// TIA Portal V17 export
// export: Created 2023-12-22T15:04:39.9681609Z, ExportSetting WithDefaults, DisplayName Totally Integrated Automation Portal, DisplayVersion V17, DisplayName TIA Portal Openness, DisplayVersion V17, DisplayName TIA Portal Version Control Interface, DisplayVersion V17, DisplayName STEP 7 Professional, DisplayVersion V17, DisplayName STEP 7 Safety, DisplayVersion V17, DisplayName WinCC Advanced, DisplayVersion V17
FUNCTION_BLOCK "AI_ex"   // FB103, LAD
{ S7_Optimized_Access := 'FALSE' }
VERSION : 0.1
// stored: AutoNumber false, IsIECCheckEnabled false, SetENOAutomatically false, UDAEnableTagReadback false
   VAR_OUTPUT
      S_Alarm : Bool;   // Внешний индикатор наличия аварии
   END_VAR
   VAR_IN_OUT
      Signal : Int;   // Входной сигнал контроллера
      Result : Real;   // Результат измерений
   END_VAR
   VAR DB_SPECIFIC
      CMD : "CMD";   // Основные команды / Блок команд
      Mode : Int;   // Режим работы
      Status : Int;   // Статус устройства
      Use : Struct   // Функционал
         RTD { S7_SetPoint := 'True'} : Bool;   // Режим RTD
         Filter { S7_SetPoint := 'True'} : Bool;   // Филтрация сигнала
         Inverse { S7_SetPoint := 'True'} : Bool;   // Инверсия сигнала
         Indirect { S7_SetPoint := 'True'} : Bool := true;   // Косвенная адресация
         Status { S7_SetPoint := 'True'} : Bool;   // Использовать подсветку
         Light { S7_SetPoint := 'True'} : Bool;   // Динамическая подсветка
         Lim_Low { S7_SetPoint := 'True'} : Bool;   // Отсечь низкие аварии
         Lim_High { S7_SetPoint := 'True'} : Bool;   // Отсечь высокие аварии
         Communication { S7_SetPoint := 'True'} : Bool;   // Передача в Value по сети
      END_STRUCT;
      VmA : Real;   // Реальный сигнал на входе ПЛК
      RTD_c { S7_SetPoint := 'True'} : Real := 10.0;   // Коэффициент RTD
      Calibration { S7_SetPoint := 'True'} : Real;   // Поправка
   END_VAR
   VAR
      Converter { S7_SetPoint := 'True'} : "Converter_LAD";   // Масштабирование сигнала
   END_VAR
   VAR DB_SPECIFIC
      SP : Struct   // Уставки аварий
         NC { S7_SetPoint := 'True'} : Real := -500.0;   // Сигнал при обрыве линии
         SC { S7_SetPoint := 'True'} : Real := 32000.0;   // Сигнал при КЗ/перегрузке
         HH { S7_SetPoint := 'True'} : Real := 90.0;   // Аварийно высокий сигнал
         H { S7_SetPoint := 'True'} : Real := 85.0;   // Высокий сигнал
         L { S7_SetPoint := 'True'} : Real := 15.0;   // Низкий сигнал
         LL { S7_SetPoint := 'True'} : Real := 10.0;   // Аварийно низкий сигнал
      END_STRUCT;
   END_VAR
   VAR
      Tx { S7_SetPoint := 'True'} : Array[0..5] of "Time_R";   // Блок таймеров
   END_VAR
   VAR DB_SPECIFIC
      Alarm : Struct   // Список аварий
         ST : Bool;   // Общая неисправность
         HH : Bool;   // сработала авария по аварийно высокму уровню
         H : Bool;   // сработало предупреждение по высокому уровню
         L : Bool;   // сработало предупреждение по низкому уровню
         LL : Bool;   // сработало предупрждение по аварийно низкому уровню
         NC : Bool;   // обрыв линии
         SC : Bool;   // короткое замыкание
      END_STRUCT;
      Alarms : Word;   // Слово аварий
      Events : Word;   // События датчика
      pos : Array[0..15] of Bool;   // Контроль фронтов событий
      Input_Type { S7_SetPoint := 'True'} : Int;   // Тип датчика, 0 - 4..20, 1 - 0..20, 2 - 0..10, 3 - 0..5, 4 - RTD
      CodeID { S7_SetPoint := 'True'} : Int;   // Код датчика для привязки в скаде
      "Type" { S7_SetPoint := 'True'} : Int;   // Тип датчика (единицы измерения)
      ADDR { S7_SetPoint := 'True'} : Int;   // Адрес входа на контроллере
      Filter_SP { S7_SetPoint := 'True'} : Int := 100;   // Ёмкость фильтра
      "Name" { S7_SetPoint := 'True'} : String[5];
   END_VAR
   VAR
      Filter_DB : "Filter";   // Фильтрация скачков сигнала
   END_VAR
   VAR DB_SPECIFIC
      Time_DTL { S7_SetPoint := 'True'} : DTL;
   END_VAR
   VAR_TEMP
      ev : Bool;   // Флаг событий
      Value : Real;   // Итоговый сигнал
      Signal_DI : DInt;   // Конвертация сигнала
      Signal_R : Real;   // Конвертация сигнала
      Type_Min : Real;
      Type_Max : Real;
   END_VAR
   VAR CONSTANT
      FALSE : Bool;
      TRUE : Bool := true;
   END_VAR
   // CMD.Start_A := true;
   // Converter.Max_In := 27648.0;
   // Converter.Max_Out := 100.0;
   VAR_TEMP   // added for the SCL form of the ladder/FBD networks
      _w1 : Bool;
      _w2 : Bool;
      _w3 : Bool;
      _w4 : Bool;
      _w5 : Bool;
      _w6 : Bool;
      _w7 : Bool;
      _w8 : Bool;
      _w9 : Bool;
      _w10 : Bool;
      _w11 : Bool;
      _w12 : Bool;
      _w13 : Bool;
      _w14 : Bool;
      _w15 : Bool;
      _w16 : Bool;
   END_VAR
BEGIN

REGION Network 1: Общий сброс
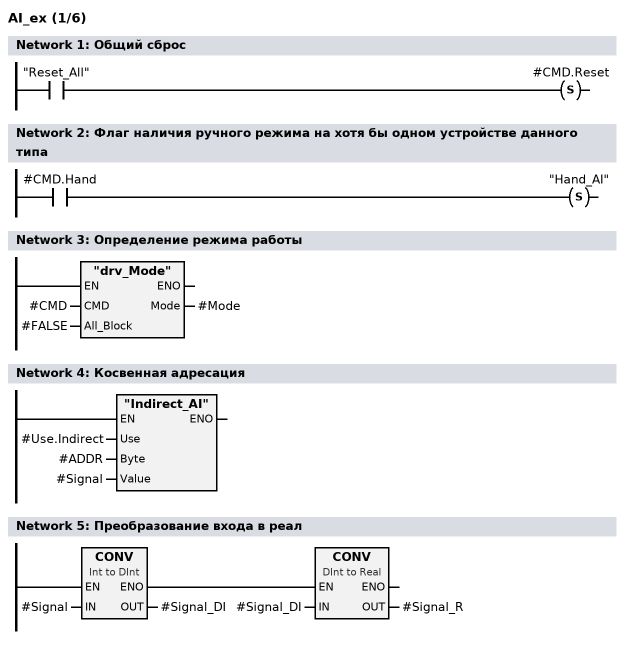
   RUNG wire#powerrail
      Contact( "Reset_All" )
      S_Coil( #CMD.Reset )
   END_RUNG
   // the same network as SCL:
   IF "Reset_All" THEN #CMD.Reset := TRUE; END_IF;
END_REGION

REGION Network 2: Флаг наличия ручного режима на хотя бы одном устройстве данного типа
   RUNG wire#powerrail
      Contact( #CMD.Hand )
      S_Coil( "Hand_AI" )
   END_RUNG
   // the same network as SCL:
   IF #CMD.Hand THEN "Hand_AI" := TRUE; END_IF;
END_REGION

REGION Network 3: Определение режима работы
   RUNG wire#powerrail
      "drv_Mode"(CMD := #CMD, All_Block := #FALSE, Mode => #Mode)
   END_RUNG
   // the same network as SCL:
   "drv_Mode"(CMD := #CMD, All_Block := #FALSE, Mode => #Mode);
END_REGION

REGION Network 4: Косвенная адресация
   RUNG wire#powerrail
      "Indirect_AI"(Use := #Use.Indirect, "Byte" := #ADDR, Value := #Signal)
   END_RUNG
   // the same network as SCL:
   "Indirect_AI"(Use := #Use.Indirect, "Byte" := #ADDR, Value := #Signal);
END_REGION

REGION Network 5: Преобразование входа в реал
   RUNG wire#powerrail
      { S7_Templates := "[SrcType := Int, DestType := DInt]"; S7_GenerateENO := "TRUE" } Convert(in := #Signal, out => #Signal_DI)
      { S7_Templates := "[SrcType := DInt, DestType := Real]"; S7_GenerateENO := "TRUE" } Convert(in := #Signal_DI, out => #Signal_R)
   END_RUNG
   // the same network as SCL:
   // ENO of a box is taken as its EN; it also drops when the box reports an error
   #Signal_DI := INT_TO_DINT(#Signal);
   #Signal_R := DINT_TO_REAL(#Signal_DI);
END_REGION

REGION Network 6: Преобразование кода в реальное значение входа
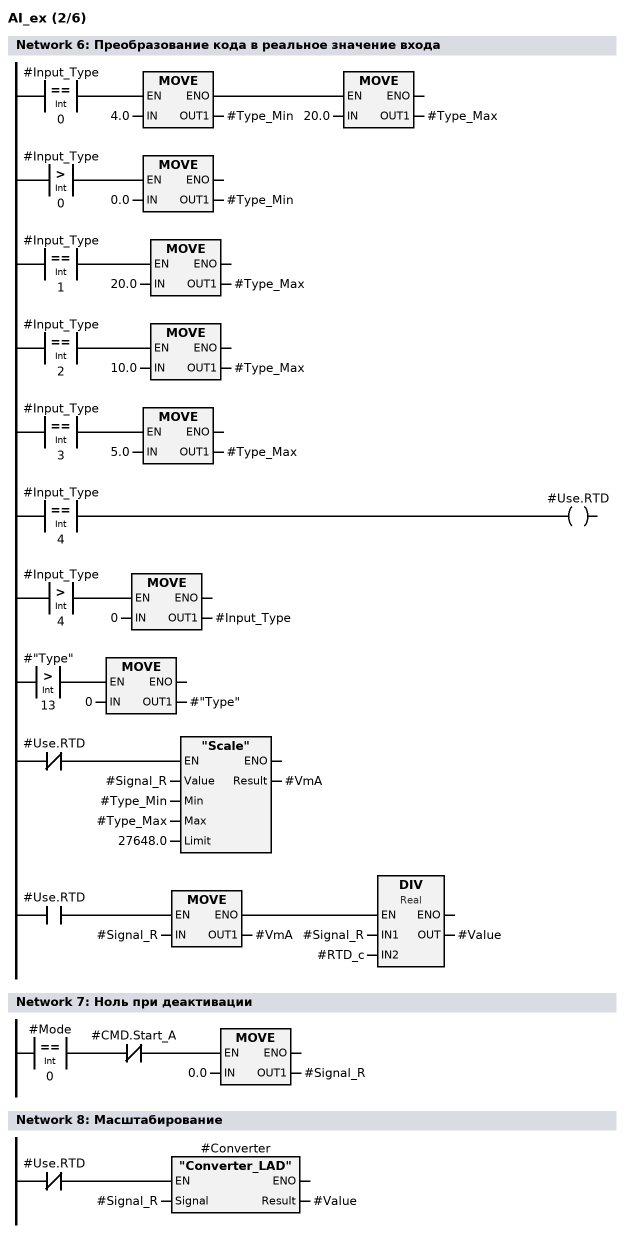
   RUNG wire#powerrail
      { S7_Templates := "SrcType := Int" } EQ_Contact(in1 := #Input_Type, in2 := 0)
      Move(in := 4.0, out1 => #Type_Min)
      Move(in := 20.0, out1 => #Type_Max)
   END_RUNG
   RUNG wire#powerrail
      { S7_Templates := "SrcType := Int" } GT_Contact(in1 := #Input_Type, in2 := 0)
      Move(in := 0.0, out1 => #Type_Min)
   END_RUNG
   RUNG wire#powerrail
      { S7_Templates := "SrcType := Int" } EQ_Contact(in1 := #Input_Type, in2 := 1)
      Move(in := 20.0, out1 => #Type_Max)
   END_RUNG
   RUNG wire#powerrail
      { S7_Templates := "SrcType := Int" } EQ_Contact(in1 := #Input_Type, in2 := 2)
      Move(in := 10.0, out1 => #Type_Max)
   END_RUNG
   RUNG wire#powerrail
      { S7_Templates := "SrcType := Int" } EQ_Contact(in1 := #Input_Type, in2 := 3)
      Move(in := 5.0, out1 => #Type_Max)
   END_RUNG
   RUNG wire#powerrail
      { S7_Templates := "SrcType := Int" } EQ_Contact(in1 := #Input_Type, in2 := 4)
      Coil( #Use.RTD )
   END_RUNG
   RUNG wire#powerrail
      { S7_Templates := "SrcType := Int" } GT_Contact(in1 := #Input_Type, in2 := 4)
      Move(in := 0, out1 => #Input_Type)
   END_RUNG
   RUNG wire#powerrail
      { S7_Templates := "SrcType := Int" } GT_Contact(in1 := #"Type", in2 := 13)
      Move(in := 0, out1 => #"Type")
   END_RUNG
   RUNG wire#powerrail
      I_Contact( #Use.RTD )
      "Scale"(Value := #Signal_R, Min := #Type_Min, Max := #Type_Max, Limit := 27648.0, Result => #VmA)
   END_RUNG
   RUNG wire#powerrail
      Contact( #Use.RTD )
      Move(in := #Signal_R, out1 => #VmA)
      { S7_Templates := "SrcType := Real"; S7_GenerateENO := "TRUE" } Div(in1 := #Signal_R, in2 := #RTD_c, out => #Value)
   END_RUNG
   // the same network as SCL:
   IF #Input_Type = 0 THEN
       #Type_Min := 4.0;
       #Type_Max := 20.0;
   END_IF;
   IF #Input_Type > 0 THEN #Type_Min := 0.0; END_IF;
   IF #Input_Type = 1 THEN #Type_Max := 20.0; END_IF;
   IF #Input_Type = 2 THEN #Type_Max := 10.0; END_IF;
   IF #Input_Type = 3 THEN #Type_Max := 5.0; END_IF;
   #Use.RTD := #Input_Type = 4;
   IF #Input_Type > 4 THEN #Input_Type := 0; END_IF;
   IF #"Type" > 13 THEN #"Type" := 0; END_IF;
   IF NOT #Use.RTD THEN
       "Scale"(Value := #Signal_R, Min := #Type_Min, Max := #Type_Max, Limit := 27648.0, Result => #VmA);
   END_IF;
   IF #Use.RTD THEN
       #VmA := #Signal_R;
       #Value := #Signal_R / #RTD_c;
   END_IF;
END_REGION

REGION Network 7: Ноль при деактивации
   RUNG wire#powerrail
      { S7_Templates := "SrcType := Int" } EQ_Contact(in1 := #Mode, in2 := 0)
      I_Contact( #CMD.Start_A )
      Move(in := 0.0, out1 => #Signal_R)
   END_RUNG
   // the same network as SCL:
   IF (#Mode = 0) AND NOT #CMD.Start_A THEN #Signal_R := 0.0; END_IF;
END_REGION

REGION Network 8: Масштабирование
   RUNG wire#powerrail
      I_Contact( #Use.RTD )
      #Converter(Signal := #Signal_R, Result => #Value)
   END_RUNG
   // the same network as SCL:
   IF NOT #Use.RTD THEN
       #Converter(Signal := #Signal_R, Result => #Value);   // "Converter_LAD"
   END_IF;
END_REGION

REGION Network 9: Вызов блока фильтрации
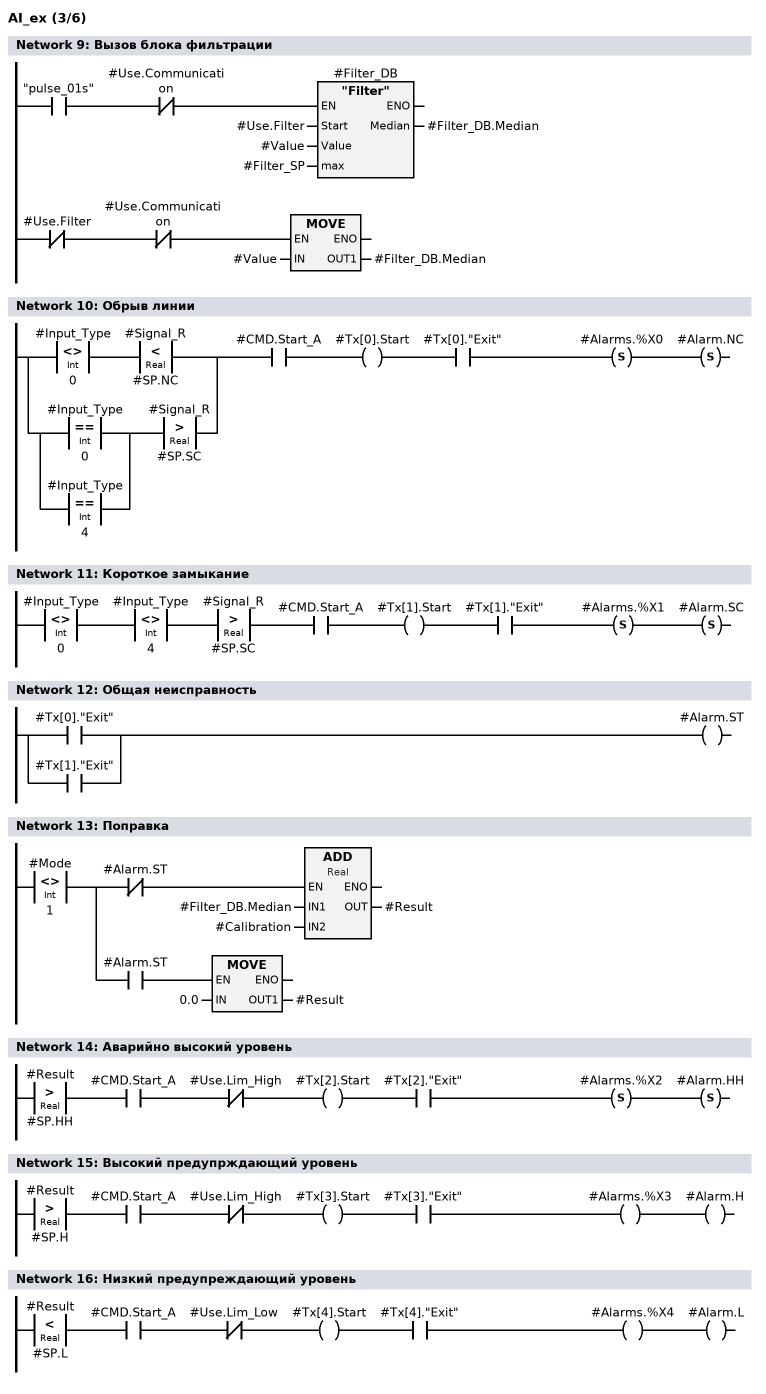
   RUNG wire#powerrail
      Contact( "pulse_01s" )
      I_Contact( #Use.Communication )
      #Filter_DB(Start := #Use.Filter, Value := #Value, max := #Filter_SP, Median => #Filter_DB.Median)
   END_RUNG
   RUNG wire#powerrail
      I_Contact( #Use.Filter )
      I_Contact( #Use.Communication )
      { S7_GenerateENO := "TRUE" } Move(in := #Value, out1 => #Filter_DB.Median)
   END_RUNG
   // the same network as SCL:
   IF "pulse_01s" AND NOT #Use.Communication THEN
       #Filter_DB(Start := #Use.Filter, Value := #Value, max := #Filter_SP, Median => #Filter_DB.Median);   // "Filter"
   END_IF;
   IF NOT #Use.Filter AND NOT #Use.Communication THEN #Filter_DB.Median := #Value; END_IF;
END_REGION

REGION Network 10: Обрыв линии
   RUNG wire#powerrail
      { S7_Templates := "SrcType := Int" } NE_Contact(in1 := #Input_Type, in2 := 0)
      { S7_Templates := "SrcType := Real" } LT_Contact(in1 := #Signal_R, in2 := #SP.NC)
      wire#w1
      Contact( #CMD.Start_A )
      Coil( #Tx[0].Start )
      Contact( #Tx[0]."Exit" )
      S_Coil( #Alarms.%X0 )
      S_Coil( #Alarm.NC )
   END_RUNG
   RUNG wire#powerrail
      { S7_Templates := "SrcType := Int" } EQ_Contact(in1 := #Input_Type, in2 := 0)
      wire#w2
      { S7_Templates := "SrcType := Real" } GT_Contact(in1 := #Signal_R, in2 := #SP.SC)
   END_RUNG wire#w1
   RUNG wire#powerrail
      { S7_Templates := "SrcType := Int" } EQ_Contact(in1 := #Input_Type, in2 := 4)
   END_RUNG wire#w2
   // the same network as SCL:
   #Tx[0].Start := (((#Input_Type <> 0) AND (#Signal_R < #SP.NC)) OR (((#Input_Type = 0) OR (#Input_Type = 4)) AND (#Signal_R > #SP.SC))) AND #CMD.Start_A;
   IF (((#Input_Type <> 0) AND (#Signal_R < #SP.NC)) OR (((#Input_Type = 0) OR (#Input_Type = 4)) AND (#Signal_R > #SP.SC))) AND #CMD.Start_A AND #Tx[0]."Exit" THEN
       #Alarms.%X0 := TRUE;
       #Alarm.NC := TRUE;
   END_IF;
END_REGION

REGION Network 11: Короткое замыкание
   RUNG wire#powerrail
      { S7_Templates := "SrcType := Int" } NE_Contact(in1 := #Input_Type, in2 := 0)
      { S7_Templates := "SrcType := Int" } NE_Contact(in1 := #Input_Type, in2 := 4)
      { S7_Templates := "SrcType := Real" } GT_Contact(in1 := #Signal_R, in2 := #SP.SC)
      Contact( #CMD.Start_A )
      Coil( #Tx[1].Start )
      Contact( #Tx[1]."Exit" )
      S_Coil( #Alarms.%X1 )
      S_Coil( #Alarm.SC )
   END_RUNG
   // the same network as SCL:
   #Tx[1].Start := (#Input_Type <> 0) AND (#Input_Type <> 4) AND (#Signal_R > #SP.SC) AND #CMD.Start_A;
   IF (#Input_Type <> 0) AND (#Input_Type <> 4) AND (#Signal_R > #SP.SC) AND #CMD.Start_A AND #Tx[1]."Exit" THEN
       #Alarms.%X1 := TRUE;
       #Alarm.SC := TRUE;
   END_IF;
END_REGION

REGION Network 12: Общая неисправность
   RUNG wire#powerrail
      Contact( #Tx[0]."Exit" )
      wire#w1
      Coil( #Alarm.ST )
   END_RUNG
   RUNG wire#powerrail
      Contact( #Tx[1]."Exit" )
   END_RUNG wire#w1
   // the same network as SCL:
   #Alarm.ST := #Tx[0]."Exit" OR #Tx[1]."Exit";
END_REGION

REGION Network 13: Поправка
   RUNG wire#powerrail
      { S7_Templates := "SrcType := Int" } NE_Contact(in1 := #Mode, in2 := 1)
      wire#w1
      I_Contact( #Alarm.ST )
      { S7_Templates := "SrcType := Real"; S7_GenerateENO := "TRUE" } Add(in1 := #Filter_DB.Median, in2 := #Calibration, out => #Result)
   END_RUNG
   RUNG wire#w1
      Contact( #Alarm.ST )
      Move(in := 0.0, out1 => #Result)
   END_RUNG
   // the same network as SCL:
   #_w1 := #Mode <> 1;
   IF #_w1 AND NOT #Alarm.ST THEN #Result := #Filter_DB.Median + #Calibration; END_IF;
   IF #_w1 AND #Alarm.ST THEN #Result := 0.0; END_IF;
END_REGION

REGION Network 14: Аварийно высокий уровень
   RUNG wire#powerrail
      { S7_Templates := "SrcType := Real" } GT_Contact(in1 := #Result, in2 := #SP.HH)
      Contact( #CMD.Start_A )
      I_Contact( #Use.Lim_High )
      Coil( #Tx[2].Start )
      Contact( #Tx[2]."Exit" )
      S_Coil( #Alarms.%X2 )
      S_Coil( #Alarm.HH )
   END_RUNG
   // the same network as SCL:
   #Tx[2].Start := (#Result > #SP.HH) AND #CMD.Start_A AND NOT #Use.Lim_High;
   IF (#Result > #SP.HH) AND #CMD.Start_A AND NOT #Use.Lim_High AND #Tx[2]."Exit" THEN
       #Alarms.%X2 := TRUE;
       #Alarm.HH := TRUE;
   END_IF;
END_REGION

REGION Network 15: Высокий предупрждающий уровень
   RUNG wire#powerrail
      { S7_Templates := "SrcType := Real" } GT_Contact(in1 := #Result, in2 := #SP.H)
      Contact( #CMD.Start_A )
      I_Contact( #Use.Lim_High )
      Coil( #Tx[3].Start )
      Contact( #Tx[3]."Exit" )
      Coil( #Alarms.%X3 )
      Coil( #Alarm.H )
   END_RUNG
   // the same network as SCL:
   #Tx[3].Start := (#Result > #SP.H) AND #CMD.Start_A AND NOT #Use.Lim_High;
   #Alarms.%X3 := (#Result > #SP.H) AND #CMD.Start_A AND NOT #Use.Lim_High AND #Tx[3]."Exit";
   #Alarm.H := #Alarms.%X3;
END_REGION

REGION Network 16: Низкий предупреждающий уровень
   RUNG wire#powerrail
      { S7_Templates := "SrcType := Real" } LT_Contact(in1 := #Result, in2 := #SP.L)
      Contact( #CMD.Start_A )
      I_Contact( #Use.Lim_Low )
      Coil( #Tx[4].Start )
      Contact( #Tx[4]."Exit" )
      Coil( #Alarms.%X4 )
      Coil( #Alarm.L )
   END_RUNG
   // the same network as SCL:
   #Tx[4].Start := (#Result < #SP.L) AND #CMD.Start_A AND NOT #Use.Lim_Low;
   #Alarms.%X4 := (#Result < #SP.L) AND #CMD.Start_A AND NOT #Use.Lim_Low AND #Tx[4]."Exit";
   #Alarm.L := #Alarms.%X4;
END_REGION

REGION Network 17: Аварийно высокий уровень
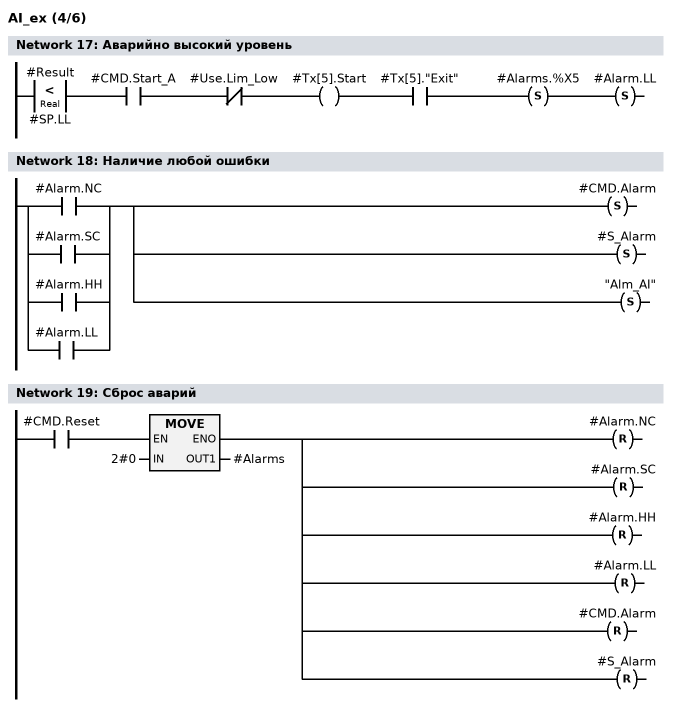
   RUNG wire#powerrail
      { S7_Templates := "SrcType := Real" } LT_Contact(in1 := #Result, in2 := #SP.LL)
      Contact( #CMD.Start_A )
      I_Contact( #Use.Lim_Low )
      Coil( #Tx[5].Start )
      Contact( #Tx[5]."Exit" )
      S_Coil( #Alarms.%X5 )
      S_Coil( #Alarm.LL )
   END_RUNG
   // the same network as SCL:
   #Tx[5].Start := (#Result < #SP.LL) AND #CMD.Start_A AND NOT #Use.Lim_Low;
   IF (#Result < #SP.LL) AND #CMD.Start_A AND NOT #Use.Lim_Low AND #Tx[5]."Exit" THEN
       #Alarms.%X5 := TRUE;
       #Alarm.LL := TRUE;
   END_IF;
END_REGION

REGION Network 18: Наличие любой ошибки
   RUNG wire#powerrail
      Contact( #Alarm.NC )
      wire#w1
      S_Coil( #CMD.Alarm )
   END_RUNG
   RUNG wire#powerrail
      Contact( #Alarm.SC )
   END_RUNG wire#w1
   RUNG wire#powerrail
      Contact( #Alarm.HH )
   END_RUNG wire#w1
   RUNG wire#powerrail
      Contact( #Alarm.LL )
   END_RUNG wire#w1
   RUNG wire#w1
      S_Coil( #S_Alarm )
   END_RUNG
   RUNG wire#w1
      S_Coil( "Alm_AI" )
   END_RUNG
   // the same network as SCL:
   IF #Alarm.NC OR #Alarm.SC OR #Alarm.HH OR #Alarm.LL THEN
       #CMD.Alarm := TRUE;
       #S_Alarm := TRUE;
       "Alm_AI" := TRUE;
   END_IF;
END_REGION

REGION Network 19: Сброс аварий
   RUNG wire#powerrail
      Contact( #CMD.Reset )
      Move(in := 2#0, out1 => #Alarms)
      wire#w1
      R_Coil( #Alarm.NC )
   END_RUNG
   RUNG wire#w1
      R_Coil( #Alarm.SC )
   END_RUNG
   RUNG wire#w1
      R_Coil( #Alarm.HH )
   END_RUNG
   RUNG wire#w1
      R_Coil( #Alarm.LL )
   END_RUNG
   RUNG wire#w1
      R_Coil( #CMD.Alarm )
   END_RUNG
   RUNG wire#w1
      R_Coil( #S_Alarm )
   END_RUNG
   // the same network as SCL:
   IF #CMD.Reset THEN
       #Alarms := 2#0;
       #Alarm.NC := FALSE;
       #Alarm.SC := FALSE;
       #Alarm.HH := FALSE;
       #Alarm.LL := FALSE;
       #CMD.Alarm := FALSE;
       #S_Alarm := FALSE;
   END_IF;
END_REGION

REGION Network 20: События датчика
   // 0 - датчик активирован
   // 1 - датчик деактивирован
   // 2 - датчик в ручном режиме
   // 3 - датчик в автоматическом режиме
   // 4 - сигнал ниже нижнего предупреждающего
   // 5 - сигнал в норме
   // 6 - сигнал выше верхнего предупреждающего
   // 7 - сигнал в норме
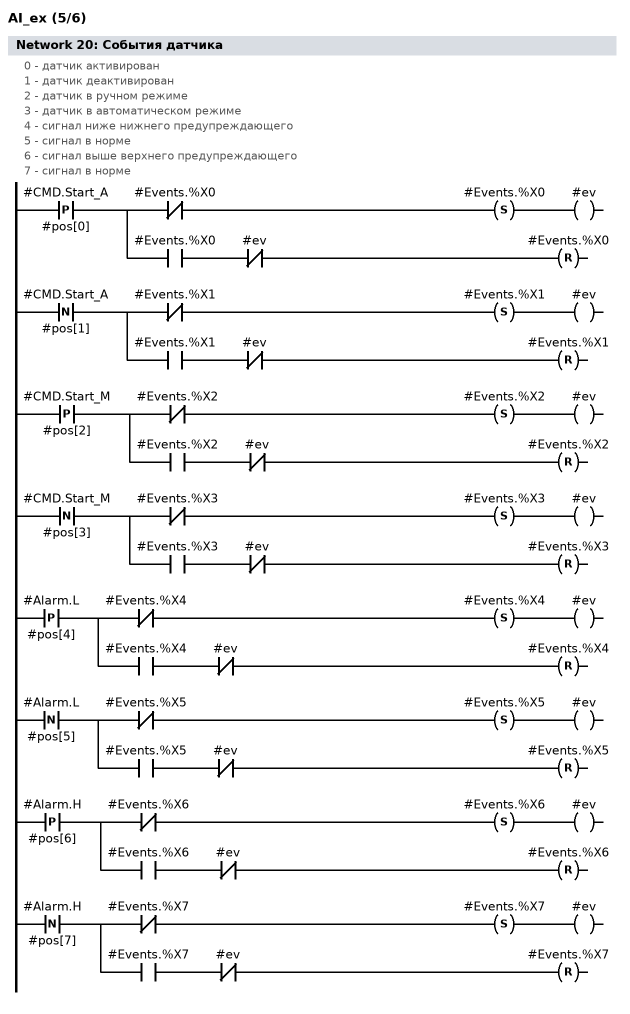
   RUNG wire#powerrail
      P_Contact(operand := #CMD.Start_A, bit := #pos[0])
      wire#w1
      I_Contact( #Events.%X0 )
      S_Coil( #Events.%X0 )
      Coil( #ev )
   END_RUNG
   RUNG wire#w1
      Contact( #Events.%X0 )
      I_Contact( #ev )
      R_Coil( #Events.%X0 )
   END_RUNG
   RUNG wire#powerrail
      N_Contact(operand := #CMD.Start_A, bit := #pos[1])
      wire#w2
      I_Contact( #Events.%X1 )
      S_Coil( #Events.%X1 )
      Coil( #ev )
   END_RUNG
   RUNG wire#w2
      Contact( #Events.%X1 )
      I_Contact( #ev )
      R_Coil( #Events.%X1 )
   END_RUNG
   RUNG wire#powerrail
      P_Contact(operand := #CMD.Start_M, bit := #pos[2])
      wire#w3
      I_Contact( #Events.%X2 )
      S_Coil( #Events.%X2 )
      Coil( #ev )
   END_RUNG
   RUNG wire#w3
      Contact( #Events.%X2 )
      I_Contact( #ev )
      R_Coil( #Events.%X2 )
   END_RUNG
   RUNG wire#powerrail
      N_Contact(operand := #CMD.Start_M, bit := #pos[3])
      wire#w4
      I_Contact( #Events.%X3 )
      S_Coil( #Events.%X3 )
      Coil( #ev )
   END_RUNG
   RUNG wire#w4
      Contact( #Events.%X3 )
      I_Contact( #ev )
      R_Coil( #Events.%X3 )
   END_RUNG
   RUNG wire#powerrail
      P_Contact(operand := #Alarm.L, bit := #pos[4])
      wire#w5
      I_Contact( #Events.%X4 )
      S_Coil( #Events.%X4 )
      Coil( #ev )
   END_RUNG
   RUNG wire#w5
      Contact( #Events.%X4 )
      I_Contact( #ev )
      R_Coil( #Events.%X4 )
   END_RUNG
   RUNG wire#powerrail
      N_Contact(operand := #Alarm.L, bit := #pos[5])
      wire#w6
      I_Contact( #Events.%X5 )
      S_Coil( #Events.%X5 )
      Coil( #ev )
   END_RUNG
   RUNG wire#w6
      Contact( #Events.%X5 )
      I_Contact( #ev )
      R_Coil( #Events.%X5 )
   END_RUNG
   RUNG wire#powerrail
      P_Contact(operand := #Alarm.H, bit := #pos[6])
      wire#w7
      I_Contact( #Events.%X6 )
      S_Coil( #Events.%X6 )
      Coil( #ev )
   END_RUNG
   RUNG wire#w7
      Contact( #Events.%X6 )
      I_Contact( #ev )
      R_Coil( #Events.%X6 )
   END_RUNG
   RUNG wire#powerrail
      N_Contact(operand := #Alarm.H, bit := #pos[7])
      wire#w8
      I_Contact( #Events.%X7 )
      S_Coil( #Events.%X7 )
      Coil( #ev )
   END_RUNG
   RUNG wire#w8
      Contact( #Events.%X7 )
      I_Contact( #ev )
      R_Coil( #Events.%X7 )
   END_RUNG
   // the same network as SCL:
   #_w1 := #CMD.Start_A AND NOT #pos[0];   // rising edge of #CMD.Start_A
   #pos[0] := #CMD.Start_A;
   #_w2 := #_w1 AND NOT #Events.%X0;
   IF #_w2 THEN #Events.%X0 := TRUE; END_IF;
   #ev := #_w2;
   IF #_w1 AND #Events.%X0 AND NOT #ev THEN #Events.%X0 := FALSE; END_IF;
   #_w3 := NOT #CMD.Start_A AND #pos[1];   // falling edge of #CMD.Start_A
   #pos[1] := #CMD.Start_A;
   #_w4 := #_w3 AND NOT #Events.%X1;
   IF #_w4 THEN #Events.%X1 := TRUE; END_IF;
   #ev := #_w4;
   IF #_w3 AND #Events.%X1 AND NOT #ev THEN #Events.%X1 := FALSE; END_IF;
   #_w5 := #CMD.Start_M AND NOT #pos[2];   // rising edge of #CMD.Start_M
   #pos[2] := #CMD.Start_M;
   #_w6 := #_w5 AND NOT #Events.%X2;
   IF #_w6 THEN #Events.%X2 := TRUE; END_IF;
   #ev := #_w6;
   IF #_w5 AND #Events.%X2 AND NOT #ev THEN #Events.%X2 := FALSE; END_IF;
   #_w7 := NOT #CMD.Start_M AND #pos[3];   // falling edge of #CMD.Start_M
   #pos[3] := #CMD.Start_M;
   #_w8 := #_w7 AND NOT #Events.%X3;
   IF #_w8 THEN #Events.%X3 := TRUE; END_IF;
   #ev := #_w8;
   IF #_w7 AND #Events.%X3 AND NOT #ev THEN #Events.%X3 := FALSE; END_IF;
   #_w9 := #Alarm.L AND NOT #pos[4];   // rising edge of #Alarm.L
   #pos[4] := #Alarm.L;
   #_w10 := #_w9 AND NOT #Events.%X4;
   IF #_w10 THEN #Events.%X4 := TRUE; END_IF;
   #ev := #_w10;
   IF #_w9 AND #Events.%X4 AND NOT #ev THEN #Events.%X4 := FALSE; END_IF;
   #_w11 := NOT #Alarm.L AND #pos[5];   // falling edge of #Alarm.L
   #pos[5] := #Alarm.L;
   #_w12 := #_w11 AND NOT #Events.%X5;
   IF #_w12 THEN #Events.%X5 := TRUE; END_IF;
   #ev := #_w12;
   IF #_w11 AND #Events.%X5 AND NOT #ev THEN #Events.%X5 := FALSE; END_IF;
   #_w13 := #Alarm.H AND NOT #pos[6];   // rising edge of #Alarm.H
   #pos[6] := #Alarm.H;
   #_w14 := #_w13 AND NOT #Events.%X6;
   IF #_w14 THEN #Events.%X6 := TRUE; END_IF;
   #ev := #_w14;
   IF #_w13 AND #Events.%X6 AND NOT #ev THEN #Events.%X6 := FALSE; END_IF;
   #_w15 := NOT #Alarm.H AND #pos[7];   // falling edge of #Alarm.H
   #pos[7] := #Alarm.H;
   #_w16 := #_w15 AND NOT #Events.%X7;
   IF #_w16 THEN #Events.%X7 := TRUE; END_IF;
   #ev := #_w16;
   IF #_w15 AND #Events.%X7 AND NOT #ev THEN #Events.%X7 := FALSE; END_IF;
END_REGION

REGION Network 21: Статус входа
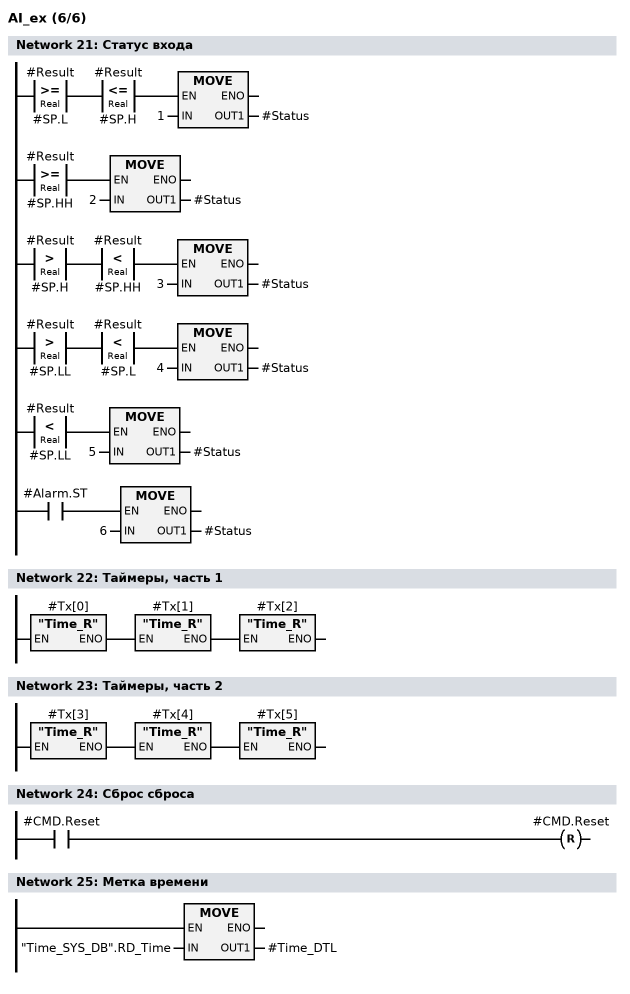
   RUNG wire#powerrail
      { S7_Templates := "SrcType := Real" } GE_Contact(in1 := #Result, in2 := #SP.L)
      { S7_Templates := "SrcType := Real" } LE_Contact(in1 := #Result, in2 := #SP.H)
      Move(in := 1, out1 => #Status)
   END_RUNG
   RUNG wire#powerrail
      { S7_Templates := "SrcType := Real" } GE_Contact(in1 := #Result, in2 := #SP.HH)
      Move(in := 2, out1 => #Status)
   END_RUNG
   RUNG wire#powerrail
      { S7_Templates := "SrcType := Real" } GT_Contact(in1 := #Result, in2 := #SP.H)
      { S7_Templates := "SrcType := Real" } LT_Contact(in1 := #Result, in2 := #SP.HH)
      Move(in := 3, out1 => #Status)
   END_RUNG
   RUNG wire#powerrail
      { S7_Templates := "SrcType := Real" } GT_Contact(in1 := #Result, in2 := #SP.LL)
      { S7_Templates := "SrcType := Real" } LT_Contact(in1 := #Result, in2 := #SP.L)
      Move(in := 4, out1 => #Status)
   END_RUNG
   RUNG wire#powerrail
      { S7_Templates := "SrcType := Real" } LT_Contact(in1 := #Result, in2 := #SP.LL)
      Move(in := 5, out1 => #Status)
   END_RUNG
   RUNG wire#powerrail
      Contact( #Alarm.ST )
      Move(in := 6, out1 => #Status)
   END_RUNG
   // the same network as SCL:
   IF (#Result >= #SP.L) AND (#Result <= #SP.H) THEN #Status := 1; END_IF;
   IF #Result >= #SP.HH THEN #Status := 2; END_IF;
   IF (#Result > #SP.H) AND (#Result < #SP.HH) THEN #Status := 3; END_IF;
   IF (#Result > #SP.LL) AND (#Result < #SP.L) THEN #Status := 4; END_IF;
   IF #Result < #SP.LL THEN #Status := 5; END_IF;
   IF #Alarm.ST THEN #Status := 6; END_IF;
END_REGION

REGION Network 22: Таймеры, часть 1
   RUNG wire#powerrail
      #Tx[0]()
      #Tx[1]()
      #Tx[2]()
   END_RUNG
   // the same network as SCL:
   #Tx[0](ENO => #_w1);   // "Time_R"
   #Tx[1](EN := #_w1, ENO => #_w2);   // "Time_R"
   IF #_w2 THEN
       #Tx[2]();   // "Time_R"
   END_IF;
END_REGION

REGION Network 23: Таймеры, часть 2
   RUNG wire#powerrail
      #Tx[3]()
      #Tx[4]()
      #Tx[5]()
   END_RUNG
   // the same network as SCL:
   #Tx[3](ENO => #_w1);   // "Time_R"
   #Tx[4](EN := #_w1, ENO => #_w2);   // "Time_R"
   IF #_w2 THEN
       #Tx[5]();   // "Time_R"
   END_IF;
END_REGION

REGION Network 24: Сброс сброса
   RUNG wire#powerrail
      Contact( #CMD.Reset )
      R_Coil( #CMD.Reset )
   END_RUNG
   // the same network as SCL:
   IF #CMD.Reset THEN #CMD.Reset := FALSE; END_IF;
END_REGION

REGION Network 25: Метка времени
   RUNG wire#powerrail
      Move(in := "Time_SYS_DB".RD_Time, out1 => #Time_DTL)
   END_RUNG
   // the same network as SCL:
   #Time_DTL := "Time_SYS_DB".RD_Time;
END_REGION
END_FUNCTION_BLOCK
